(* CODESYS project GPS.4g.20210713.1.project

Project tree, tasks and I/O mapping:
  MIC7001 : Changsha-Cyber-MI-linux, Changsha Cyber-MI Co., Ltd., version 3.5.10.40
    application Application
      libraries: Standard, * (System); CAA Types Extern, * (CAA Technical Workgroup); CAA Callback Extern, * (CAA Technical Workgroup); SysMem, * (System); SysTypes Interfaces, * (System); SysTime, * (System); CAA DTUtil Extern, 3.5.12.0 (CAA Technical Workgroup); CAA Real Time Clock Extern, 3.5.10.0 (CAA Technical Workgroup); CAN API, 1.0.0.3 (3S - Smart Software Solutions GmbH); SysFile, 3.5.15.0 (System); AC_DataLog, 3.5.14.0 (3S - Smart Software Solutions GmbH); CAA Net Base Services, 3.5.15.0 (CAA Technical Workgroup); CAA Memory, 3.5.12.0 (CAA Technical Workgroup); CAA SerialCom, 3.5.15.0 (CAA Technical Workgroup); Util, 3.5.15.0 (System); CAA Can Low Level Imp Extern, 3.5.11.0 (CAA Technical Workgroup); CAA Can Low Level Extern, 3.5.15.0 (CAA Technical Workgroup); VisuDialogs, * (System); CmpBitmapPool, * (System); CAA File, 3.5.15.0 (CAA Technical Workgroup); IODrvEtherCAT, 3.5.15.50 (3S - Smart Software Solutions GmbH); SysShm Implementation, 3.5.16.0 (System); SysShm, 3.5.8.0 (System); MIC7001 base library, 1.11 (Cyber-MI.com)
      task VISU_TASK (cyclic, interval 100 ms, priority 31) calls prg_gps, VisuElems.Visu_Prg
      10_gvls/
        global variables gvl_remoter
        global variables GVL_prg_weight
        global variables GVL_IO
        global variables GVL_ES
        global variables GVL
        global variables GVL_can
        global variables GVL_par
      06_jt808/
        programs/
          program prg_gps [ST]
          program prg_jt808 [ST]: send_to_server, read_from_server, init
        Structs/
          data type stShmJT808Down
          data type stLocationExt
          data type stShmJT808Up
          data type stLocationBase
          data type stCanFrm
          data type nmeaTIME
          data type nmeaGPRMC
        functionblocks/
          function block Com_gps [ST]
        functions/
          function get_sub_string_1 [ST]
          function nmea_parse_time [ST]
          function nmea_parse_date [ST]
          function get_latlon_from_str [ST]
          function nmea_parse_GPRMC [ST]
    SoftMotion General Axis Pool
  libraries: CmpBitmapPool, * (System)
  5ce3da45-db07-42e7-a21c-a00fff4ed8f6|D:\工作文件\009中集集团\DOCS\等油耗图.jpg
  5ce3da45-db07-42e7-a21c-a00fff4ed8f6|C:\Users\RJST\Desktop\bmp1.png
  text list GlobalTextList
*)

// MIC7001/Application/06_jt808/Structs/stShmJT808Down
TYPE stShmJT808Down :  // JT808下行数据
STRUCT
	location_interval:DINT;  // 位置信息发送间隔， 单位： ms
	ctrl : DINT;   // 车辆控制命令
END_STRUCT
END_TYPE

// MIC7001/Application/06_jt808/Structs/stLocationExt
TYPE stLocationExt :
STRUCT
	km_all: DINT;  // km all
	fuel:INT;   // fuel meter
	speed: INT;  // speed can
	lac:DINT; 
	cid:DINT;
	fuel_trip:DINT; // 本行程油耗
	fuel_all:DINT; 
	fuel_r_h:DINT;  // 0.05L/h
	fuel_r_l:DINT;  //  1/512Km/L
END_STRUCT
END_TYPE

// MIC7001/Application/06_jt808/Structs/stShmJT808Up
TYPE stShmJT808Up :   // 发送到服务器的上行数据
STRUCT
    location:stLocationBase;
	loc_ext:stLocationExt;
	can_data:stCanFrm;
END_STRUCT
END_TYPE

// MIC7001/Application/06_jt808/Structs/stLocationBase
TYPE stLocationBase :
STRUCT
	warning : UDINT;
    status : UDINT;
    latitude : DINT;
    longitude : DINT;
    altitude : INT;
    speed : INT;
    bearing : INT;
    asc_time :ARRAY[0..5] OF BYTE;  // ascii YYMMDDhhmmss (GMT+8)
END_STRUCT
END_TYPE

// MIC7001/Application/06_jt808/Structs/stCanFrm
TYPE stCanFrm :
STRUCT
	sn:UDINT;  // 每次更新内容后加一，用于通知底层发送程序
	id:UDINT;  //  CAN id
	data:ARRAY[0..7] OF BYTE;  // 8个字节 数据
END_STRUCT
END_TYPE

// MIC7001/Application/06_jt808/Structs/nmeaTIME
TYPE nmeaTIME :
STRUCT
	year:DINT;
	month:DINT;
	day:DINT;
	hour:DINT;
	minute:DINT;
	second:DINT;
	hsecond:DINT;
END_STRUCT
END_TYPE

// MIC7001/Application/06_jt808/Structs/nmeaGPRMC
TYPE nmeaGPRMC :
STRUCT
	utc : nmeaTIME;
	status : STRING(1);
	lat : REAL;
	ns : STRING(1);
	lon : REAL;
	ew : STRING(1);
	speed : REAL;
	direction : REAL;
	declination : REAL;
	declin_ew : STRING(1);
	mode : STRING(1);
END_STRUCT
END_TYPE

// MIC7001/Application/10_gvls/gvl_remoter
{attribute 'qualified_only'}
VAR_GLOBAL
    // byte0
    link:DINT;   //连接状态
    acc: BOOL ;  // 加速
    dec:BOOL ;   // 减速
    mix:BOOL;    // 搅拌
    dump:BOOL;   // 卸料
    
    // byte1
    up:BOOL;     // 
    down:BOOL;
    left:BOOL;
    right:BOOL;
    auto_add_water:BOOL;
    e_stop:BOOL;  // 急停按钮
    
    // byte2
    
END_VAR

// MIC7001/Application/10_gvls/GVL_prg_weight
{attribute 'qualified_only'}
VAR_GLOBAL
	
weight_01,weight_02,weight_03:REAL:=0;

weight_load_01,weight_load_02,weight_load_03:REAL:=0;

net_weight:REAL:=0;


ad_load	 :REAL; 
SET_load1   :REAL;  	//设定重量 砝码1
SET_load2   :REAL;	//设定重量 砝码2
SET_load3 	:REAL;		//设定重量 砝码3
SET_load4   :REAL;  	//设定重量 砝码1
SET_load5   :REAL;	//设定重量 砝码2
SET_load6 	:REAL;		//设定重量 砝码3

load_up1    :REAL;	//标定的提升重量 1
load_up2   :REAL;		//标定的提升重量 2
load_up3 	:REAL;;		//标定的提升重量 3
load_up4    :REAL;	//标定的提升重量 1
load_up5   :REAL;		//标定的提升重量 2
load_up6 	:REAL;;		//标定的提升重量 3


AD_load_up1    :REAL;
AD_load_up2    :REAL;
AD_load_up3    :REAL;
AD_load_up4    :REAL;
AD_load_up5    :REAL;
AD_load_up6    :REAL;


END_VAR

// MIC7001/Application/10_gvls/GVL_IO
{attribute 'qualified_only'}
VAR_GLOBAL

AI_curr_a				:   DWORD ;   	// 电磁阀电流A
AI_curr_b				:   DWORD ;   	// 电磁阀电流B

Putter_position			:   DWORD ;     // C17推杆位置
A_three_load			:	DWORD;		// C29 三态开关信号

AI_F_Tank_speed_set		:   DWORD ;  	//	C31 /角位移 前面罐速设定
AI_BL_Tank_speed_set	:   DWORD ;   	//  C19 后左罐速设定
AI_BR_Tank_speed_set	:   DWORD ;   	//  C20后右罐速设定

Joystick				:	DINT;   // 操纵杆 角位移
set_speed_Tank			:	REAL;	//设定罐子速度
Joystick_min			:	DINT:=2020 ; 	//小值
Joystick_mid			:	DINT :=2405; 	//中值
Joystick_max			:	DINT :=2642; 	//最大值



set_speed_temp_tank		:	real;	// 设定罐速

VCC						:   DWORD ;		//控制电压
VCC_L					:   DWORD ;		//系统电流
A_REMOTe_youmen			:   DWORD ;		//远程油门
out5v			:   DWORD ;		//输出5V 
AI_Putter_position_feedbake	:   DWORD:=0 ;		// C17 阀推杆位置反馈


// out 
bforeward_Direction		:	BOOL;		//C03 搅动指示 
bRevers_Direction		:	BOOL;		// C01 出料状态指示灯 
 
out_tor_grade_k1		:BOOL;		 	//  C25  中载  多态输出K1
out_tor_grade_k2		:BOOL; 			//  C24	 轻载 多态输出K2

hb_pwm_L				:DWORD:=0;		//  C08电机正转 输出电流
hb_do_L					:BOOL:=FALSE;	//  C23电机正转 H桥低有效

hb_pwm_R				:DWORD:=0;		//  C09电机反转 输出电流
hb_do_R					:BOOL:=FALSE;	//  C35电机反转  H桥低有效
	
/////////////////////////
pwmForward 				: DWORD;  		// 
pwmRevers 				: DWORD;  	 	// 

Pump_foreward			:	DWORD ;     // 泵比例1 正转
Pump_Revers			:	DWORD;  // 泵比例2 反转
Throttle 		:	DWORD;   // 远程油门  0.3 ~ 1.9V
Throttle2 		:	DWORD;   // 远程油门 2 倍  0.6 ~ 3.8V






//Tank_dir			:	BOOL;  //计数 A
Tank_Speed_count		:	DWORD;  //计数 B
//bWater_washlimt	: 	BOOL; // 摆杆限位 

PI02_A,PI03_B:DWORD;		//接近开关计数
PI00,PI01,PI02,PI03	:DWORD;	//接近开关计数

DI02_A,DI03_B	: 	BOOL; 	//接近开关电平



lagan_foreward_Direction		:	BOOL;	//拉杆搅动
lagan_Revers_Direction		:	BOOL;	// 拉杆 卸料

//b_foreward_Direction	:	BOOL;	//搅驾驶室操作搅动
//b_Revers_Direction		:	BOOL;	//驾驶室操作 卸料




remote_di :BOOL := FALSE; //绑定变量 驾驶室开关， 为True则通过遥控方式控制罐体， 不使用拉杆
b_mode_remote : BOOL  := FALSE;  // 驾驶室开关， 为True则通过遥控方式控制罐体， 不使用拉杆


SET_Putter_position:DINT;	//推杆位置 换算
Putter_avg:	DINT;		//推杆位置 
Putter_mid_dema:	DINT;//推杆中位标定
Putter_position_ERR,Joystick_ERR,J1939_ERR	:BOOL; //角位移，电机位置反馈  故障指示
flag_stir_enable:BOOL	;//允许搅动状态位
flag_Constant_speed:BOOL	;// 不允许 卸料 标志位 

//处理之后的数值

temp_Hydraulic_oil:REAL;	//油温值
Dprss_pumpA		:REAL; 		//正转马达压力值
Dprss_pumpB		:REAL; 		//反转马达压力值
Dprss_Water		:REAL;		//清洗水压
Dwater_level	:REAL;		//水位

iPump_foreward		:	REAL;   // 泵比例正向 
iPump_Revers 		:	REAL;  	// 泵比例反向
itank_dir            :DINT;
iPump_PID            :REAL;
END_VAR

// MIC7001/Application/10_gvls/GVL_ES
{attribute 'qualified_only'}
VAR_GLOBAL
	// send to cloud my mqtt	
	working_mode:UINT;  // 工作模式 0:熄火停车， 1：空车等待， 2：正在装料， 3：满车行驶，4：满车等待，5：正在卸料， 6：空车行驶
	rpm_engine:DINT; // 发动机转速  转/分
	rpm_set :DINT ;  // 设定发动机转速 转/分
	power_engine:REAL; // 发动机功率 千瓦
	torque_engine:REAL;// 发动机扭矩 牛米
	fuelrate_engine:REAL;// 发动机瞬时油耗 升/小时
	effect_engine:REAL;// 发动机瞬时效率 %
	fuelall_engine:REAL;// 发动机累计油耗 升
	loadrate_engine:REAL;// 发动机负载率 %
	hours_engine:REAL;// 发动机工作时间  小时
	press_pump:REAL; // A B 口压力差
	press_pump_a:REAL;// 油泵主压 A 兆帕
	press_pump_b:REAL;// 油泵主压 B 兆帕
	dir_pump:DINT;// 油泵方向 1：正转， 0： 停止，  -1：反转
	curr_a_pump:REAL;//  油泵电流A  毫安
	curr_b_pump:REAL;//  油泵电流B  毫安
	power_pump:REAL;// 油泵输出功率 千瓦
	swept_pump:REAL;// 油泵排量 毫升/转
	flow_pump:REAL;// 油泵流量 升/分
	effect_pump:REAL;// 油泵效率 %
	torque_pump:REAL;// 油泵扭矩 牛米
	dir_tank:DINT;// 搅拌桶方向 1：正转， 0： 停止，  -1：反转
	rpm_tank:REAL;// 搅拌桶转速 转/分
	weight_tank:REAL;// 搅拌桶重量 吨
	power_tank:REAL;// 搅拌桶功率 千瓦
	effect_tank:REAL;// 搅拌桶效率 %
	torque_tank:REAL;// 搅拌桶扭矩 牛米
	volume:REAL;// 当前方量 立方米
	volume_all:REAL;// 累计方量 立方米
	mileage_all:REAL;// 累计里程 千米
	grade_gear:DINT;// 变速箱档位
	rate_gear:REAL;// 变速箱变比
	rpm_gear:REAL;// 变速箱输出转速 转/分
	torque_gear:REAL;// 变速箱输入扭矩 牛米
	power_gear:REAL;// 变速箱输出功率 千瓦
	effect_gear:REAL;// 变速箱效率 %
	weight_all:REAL;// 整车重量 吨
	speed:REAL;   // 行车速度 Km/h
	power_running:REAL;  // 行车功率 Kw
	acc_running:REAL; // 行车加速度 Km/h/s
	fuel_trip_engine:REAL;  // 行程总油耗
	torque_grade:DINT;  // 节能模式： 0：轻载， 1： 中载，  2：重载
	acc_pad : REAL;  // 油门踏板 百分比
	fuel_wait:REAL :=0;  // 本行程等待油耗 L
    time_wait:REAL := 0;  // 本行程等待时间 s
    fast_acc_cntr :DINT := 0; // 急加速次数
    fast_dec_cntr :DINT := 0; // 急刹车次数
    low_grade_cntr:DINT := 0; // 低档高速次数
	fuel_100km:REAL;  // 百公里油耗
    fuel_level:REAL;  // 油耗水平 0~100
	Engine_Hour:REAL;
	
	trip_all_1939:REAL;    // 里程累计
	trip_curr_1939:REAL;  // 里程小计

	trip_all_1939_2:REAL;    // 里程累计, 高分辨率
	trip_curr_1939_2:REAL;  // 里程小计, 高分辨率
	
	temp_coolant_1939:DINT;
	Eng_Fuel_Temp:DINT;
	Eng_Oil_Temp:DINT;
	Turbo_Oil_Temp:DINT;
	Eng_InterCooler_Temp:DINT;
	Eng_InterCooler_Thermostat_Opening:DINT;
	oil_press_1939:REAL;
	coolant_level_1939:REAL;
	acc_set:BYTE;
    
    rpm_disp:ARRAY[0..9999] OF DINT;
    tor_disp:ARRAY[0..9999] OF DINT;
    ptr_disp:DINT  := 0;
    x:DINT;
    y:DINT;
    z:DINT;
	grade_joystick:REAL := 0;  // 1~10
	
	shift:DINT;  // 离合
	brake:DINT;  // 刹车
END_VAR

VAR_GLOBAL CONSTANT
	retain_max : DINT := MIC7001_BASE.Constants.RETAIN_NUM_MAX;
	// 柴油机扭矩曲线
	rpm_in:ARRAY[0..255] OF REAL := [700, 800,  900,  1000, 1100, 1200, 1300, 1400, 1500, 1600, 1700, 1800, 1900, 2000, 2100];
 	tor_h:ARRAY[0..255] OF REAL :=  [922, 1100, 1350, 1488, 1600, 1600, 1600, 1600, 1570, 1495, 1410, 1320, 1221, 970,  555];
	tor_m:ARRAY[0..255] OF REAL :=  [922, 1100, 1350, 1488, 1600, 1550, 1480, 1350, 1200, 1000,  750, 0,     0,   0,    0];
 	tor_l:ARRAY[0..255] OF REAL :=  [922, 1100, 1200, 1020, 800,  620,  460,  320,  200,  100,   0,   0,     0,   0,    0];	
END_VAR

// MIC7001/Application/10_gvls/GVL
VAR_GLOBAL CONSTANT
	retain_max : DINT := MIC7001_BASE.Constants.RETAIN_NUM_MAX;
END_VAR

VAR_GLOBAL
	
	flag_mode:bool;
	bTank_wash_Fnish:BOOL;
	
	xEnaSE:BOOL := TRUE;  // 启用节能模式
	xEnaLowRPM:BOOL := TRUE;  // 启用起步降速功能
	xEnaTor :BOOL := TRUE;  // 启用扭矩调节功能
	
	//熟数据
	g_ai_press_pump : REAL;  // 油泵主压， 单位： MPa	
	
	falg_tank_control,flag_chute_control,flag_Clean_control:BOOL;
	
	//
	g_uiYear:UINT := 1970;
	g_uiMonth:UINT := 1;
	g_uiDate:UINT := 1;
	g_uiHour:UINT := 0;
	g_uiMinute:UINT := 0;
	g_uiSecond:UINT := 0;
	
	//小时计相关
	g_running_mins:DINT := 0; //控制器运行的分钟数  retain
	g_engine_mins:DINT := 0; //发动机运行的分钟数   retain
	
	g_engine_mins_1_start:DINT := 0; //阶段小时计1开始时间  retain
	g_engine_mins_2_start:DINT := 0; //阶段小时计2开始时间  retain

	g_engine_mins_1:DINT := 0;  //发动机运行分钟数  阶段1 
	g_engine_mins_2:DINT := 0;  //发动机运行分钟数  阶段2
	
	// PORT CAN1 GLOBAL HANDLE
	g_hCan1939: CAA.HANDLE ;
	g_hRecv_FEEE: CAA.HANDLE := 0;
	g_hRecv_FEEF: CAA.HANDLE := 0;
	g_hRecv_F003: CAA.HANDLE := 0;
	g_hRecv_F004: CAA.HANDLE := 0;
	g_hRecv_18F: CAA.HANDLE := 0;
	
	//发动机相关实时数据
	g_P_KW_max:DINT := 30;  //当前发动机储备功率
	g_rpm_set: DINT := 1000;  //当前设定转速
	g_rpm_real: DINT := 0; //当前实时转速
	g_fuel_rate_1939:REAL := 0; //从发动机读到的瞬时油耗，单位：ml/s
	g_temp_coolant_1939:REAL := 0; //从发动机读到的水温， 单位：摄氏度
	g_flag_coolant_high:bool := false;  //水温报警标志
	g_oil_press_1939:REAL := 0; //从发动机读到的机油压力， 单位： kPa
	g_coolant_level_1939:REAL := 0; //从发动机读到的冷却液液位， 单位： 百分比
	g_load_percent_1939:REAL := 0; //从发动机读到的发动机负载率， 单位： 百分比
	g_demand_torque_1939:DINT := 0; //从发动机读到的需求扭矩， 单位： 百分比
	g_real_torque_1939:DINT := 0; //从发动机读到的实际扭矩， 单位：百分比
	g_acc_1939: BYTE := 0;  //从发动机读到的油门踏板百分比
	g_perfect_rpm: DINT := 0;  //从发动机读到的当前理想转速，单位 ：rpm
	g_tor_idle_1939: BYTE := 0;  //从发动机读到的当前摩擦转矩，单位：百分比
	g_real_torque_nm_1939: DINT := 0;
	g_working_old:BOOL := FALSE;
//动态调整参数	


	g_acc_set :BYTE := 40;   //需要设置的油门踏板百分比
	g_tor_set :BYTE := 1;   //需要设置的扭矩曲线号
	g_droop_set :BYTE := 16#F0;   //设置调速率

	rpm_lost_point:DINT := 50;
	
	g_x_duty_max :REAL := 70;	
	g_x_duty_min :REAL := 60;
	g_x_rpm_up_step: INT := 5;
	g_x_rpm_down_step: INT := 1;
	
	g_x_tor_max:REAL := 90;
	g_x_tor_min:REAL := 70;
	g_x_pump_up_step: INT := 1;
	g_x_pump_down_step: INT := 2;
	
	g_enable_rpm_adj:BOOL := TRUE;
	

	//retain paras 
	g_retain_01:ARRAY[0..retain_max] OF DINT;
	g_retain_02:ARRAY[0..retain_max] OF DINT;
	g_mins:ARRAY[0..MIC7001_BASE.Constants.RETAIN_NUM_MAX] OF DINT;
//动态调整参数	
	
	//统计数据
	g_fuel_depleted : DINT := 0;  //出厂累计油耗，单位：毫升
	g_fuel_depleted_1: DINT := 0; //阶段一累计油耗，单位：毫升
	g_fuel_depleted_2: DINT := 0; //阶段二累计油耗，单位：毫升
	
	g_Eng_Coolaant_Temp:INT;(*spn 110*)
	g_Eng_Fuel_Temp:INT;(*spn 174*)
	g_Eng_Oil_Temp:INT;(*spn 175*)
	g_Turbo_Oil_Temp:INT;(*spn 176*)
	g_Eng_InterCooler_Temp:INT;(*spn 52*)
	g_Eng_InterCooler_Thermostat_Opening:BYTE;(*spn 1134*)
	
						
	g_res_prop:REAL := 20; //电磁比例阀电阻，动态调整

	g_ai_pilot:REAL;
	g_ai_pilot_trace: REAL;
	g_ai_curr_prop:UINT;
	g_ai_curr_prop_trace:REAL;
	g_ai_oil_water:BOOL;
	g_ai_vcc:DWORD;
	g_ai_fuel_level:REAL;

	g_di_start:BOOL := FALSE; //上电信号
	g_di_move:BOOL := FALSE; //工作装置压力开关
	g_di_work:BOOL := FALSE; //行走压力开关
	g_di_pilot:BOOL := FALSE;  //先导手柄开关输入
	
	g_do_start:BOOL := TRUE;  //启动继电器		
	g_do_ecu:BOOL := TRUE;    //为true为发动机ECU供电
	g_do_pilot:BOOL := FALSE;
	
	g_pwm_prop:DINT := 0; 
	
	g_rpm_trace:REAL := 0;  //示波器变量，转换到0~10之间
	//间接计算数据
	g_psp: REAL := 0;   //电磁比例阀二次压力  MPa
	g_backup_power:REAL := 0;   //发动机储备功率  KW
	g_backup_power_trace:REAL; //示波器变量，转换到0~10之间
	g_duty_power:REAL := 0; //发动机功率利用率
	g_backup_torque:REAL := 0;  //发动机储备扭矩  N*M
	g_backup_torque_trace:REAL;//示波器变量，转换到0~10之间
	g_duty_torque:REAL := 0;  //发动机扭矩利用率
	g_flow1 :REAL := 0;   //前泵流量 L/min
	g_flow1_trace:REAL;//示波器变量，转换到0~10之间
	g_flow2 :REAL := 0;   //后泵流量 L/min
	g_flow2_trace:REAL;//示波器变量，转换到0~10之间
	g_power_pump1 :REAL := 0;   //前泵功率  KW
	g_power_pump1_trace:REAL;//示波器变量，转换到0~10之间
	g_power_pump2 :REAL := 0;   //后泵功率  KW
	g_power_pump2_trace:REAL;//示波器变量，转换到0~10之间
	g_torque_pump1 :REAL := 0;  //前泵输出扭矩  N*M
	g_torque_pump2 :REAL := 0;  //后泵输出扭矩  N*M
	
// I/O port mapping var
	AI_pump1:DWORD; //前泵压力
	AI_pump2:DWORD; //后泵压力
	AI_pilot:DWORD; //先导压力
	AI_curr_prop:DWORD; //电磁比例阀电流
	AI_oil_water:DWORD; //油水分离器
	AI_vcc:DWORD; //电源电压 mV
	AI_grade:DWORD; //油门旋钮
	AI_temp_oil:DWORD; //液压油温
	AI_fuel_level:DWORD; //液位传感器
	AI_idle_button:dword; //机械怠速按钮
	
	DI_start: BOOL; //启动信号
	DI_pilot:BOOL; //先导手柄闭合
	DI_move:BOOL; //行走压力开关
	DI_work:BOOL; //作业压力开关
	DI_air_filter:BOOL;  //空滤堵塞
	DI_idle_button:BOOL;  //机械怠速按钮
	DI_high_power:BOOL; //增力信号输入
	
	DO_start: BOOL := FALSE; //驱动启动电机
	DO_stop: BOOL := TRUE;  //驱动熄火继电器
	DO_pilot :BOOL := TRUE;  //驱动先导阀
	DO_high_power:BOOL := FALSE; //增力输出
	DO_high_speed:BOOL := FALSE; //高速输出
	DO_dump_load:BOOL := FALSE; //卸载输出
						
	PWM_prop:DWORD; //油泵电磁比例阀	
	
	RPM_engine:UINT; //柴油机转速  J1939

	DO_led_run:BOOL;
	DO_led_err:BOOL;
	DO_led_usr:BOOL;
	
// 档位校准	
	adj_gear: BOOL := FALSE;  //校准档位旋钮
	gear_grade: UINT := 1;   //档位旋钮对应的档位
	running_grade:DINT := 1;  //当前实际运行的档位
	
	g_grade: DINT;	  //发动机档位
	//各档位对应的转速

	g_running_grade_x:DINT := 1;
	g_power_avg_num: DINT := 10;  // 200 ms
	g_method_mode_A :DINT := 0;   // 0: based power_avg;   1: based load1939
	g_overpress_time:DINT := 100;   //1 second
	
//显示屏发送来的命令
//	cmd_auto_idle : BOOL := TRUE;
//	cmd_high_speed: BOOL := FALSE;	
//	cmd_more_power: BOOL := FALSE;
//	cmd_clear_hours : BOOL := FALSE;
//	cmd_clear_hours_1 :BOOL := FALSE;
//	cmd_clear_hours_2 :BOOL := FALSE;
	
	g_time_good: BOOL := FALSE;  //控制器本地时钟校准完成
	g_working: BOOL := false;
	g_err_fuel_level: BOOL;
	g_fuel_level: DINT;
	adj_1: BOOL;
	adj_10: BOOL;
	
	rpm_lost_rate: REAL;
	g_err_temp_oil: BOOL;
	g_temp_oil: DINT := 0;


	
	g_duty_power_avg: REAL := 0;
	g_duty_torque_avg: REAL;

	g_x_power_avg: REAL := 0;
	g_x_dest_grade: DINT := 1;
	g_torque_engine: REAL := 0;
	g_power_engine: REAL := 0;
	mode_a_up: DINT := 90;   // %
	mode_a_down:DINT := 80;  // %
	g_press12_avg: REAL := 0;
	g_press12_avg_all: REAL := 0;
	g_fuel_all_1939: DINT := 0;
	g_fuel_all: DINT := 0;
	
	g_lock_flag:BOOL := FALSE;
	g_lock_level:DINT := 0;
	gps_lock_h: BOOL := FALSE;
	gps_lock_s: BOOL := FALSE;
	gps_lock_l: BOOL := FALSE;
	
	need_send_mid :ARRAY[16#507..16#520] OF BOOL;
	need_ack_mid :ARRAY[16#307..16#320] OF BOOL;
	got_ack_mid :ARRAY[16#307..16#320] OF BOOL;
	
END_VAR




(*end of var_global for mqtt *****************************************************)


VAR_GLOBAL CONSTANT
	inmode_file:STRING:='/userapp/PlcLogic/in_mode.txt';
	mins_file :STRING := '/userapp/r_mins.txt';
END_VAR

// MIC7001/Application/10_gvls/GVL_can
{attribute 'qualified_only'}
VAR_GLOBAL
	
//can_send

	g_acc_set:BYTE;
	g_tor_set:BYTE; //扭矩曲线选择，0对应最高，2对应最低
	g_droop_set:BYTE;

	CansendData_18FF01FF : ARRAY[0..7] OF BYTE;     //系统传感器ID（搅拌车）0x18FF01FF  T 100ms   控制器发送 	
	
	CansendData_18FF02FF : ARRAY[0..7] OF BYTE;     //系统传感器ID（搅拌车）0x18FF01FF  T 100ms   控制器发送 	
	CansendData_18FF03FF : ARRAY[0..7] OF BYTE;     //系统传感器ID（搅拌车）0x18FF01FF  T 100ms   控制器发送 	
	
	CansendData_18FF66FF : ARRAY[0..7] OF BYTE;     //智能自动化控制器ID1（搅拌车）	0x18FF66FF	65280	6	Periodic	500 SEND 
	CansendData_18FF68FF : ARRAY[0..7] OF BYTE;  //智能自动化控制器报警ID1（搅拌车）	0x18FF68FF	65280	6	Periodic	500ms

	
	
	LoadingWashST,UnloadingWashReqST :BOOL;
	AutoClearWaterReqST:BOOL;
	AutoAddWaterReqST:BOOL;
	TankWashReqST:BOOL;
//can_receive
	
	CanReadData_18FF46FF : ARRAY[0..7] OF BYTE; 	//塌落度 ID 0x18FF46FF   T 500ms   网关发送 	
	CanReadData_18FF61FF : ARRAY[0..7] OF BYTE; 	//胎压传感器数据帧ID 0x18FF61FF  T 250ms   网关发送    暂不接收和转发
	CanReadData_18FF62FF : ARRAY[0..7] OF BYTE; 	//自动充气ID 0x18FF62FF   T 250ms   网关发送    暂不接收和转发	
	CanReadData_18FF64FF : ARRAY[0..7] OF BYTE;		//集中润滑ID	0x18FF64FF	65280	6	Periodic	500  网关发送    暂不接收和转发
	CanReadData_18FF6AFF : ARRAY[0..7] OF BYTE;		//GW_AdasInputs2	ADAS系统输入信息  ID2	0x18FF6AFF	65280	6	Periodic	100 网关  无用
	
	CanReadData_18FF01FE : ARRAY[0..7] OF BYTE;		//HU_ControlInformation1	大屏 ID1	0x18FF01FE	65280	6	Periodic	100	8  
	CanReadData_18FF02FE : ARRAY[0..7] OF BYTE;		//HU_ControlInformation2	大屏ID2		0x18FF02FE	65280	6	Periodic	100ms	8  FROM 显示屏据
	CanReadData_18FF03FE : ARRAY[0..7] OF BYTE;		//HU_ControlInformation2	大屏ID3		0x18FF03FE	65280	6	Periodic	100ms 	8  FROM 显示屏据

demo_cntr:UINT := 0;

// 控制器发送到操作面板数据 0x18ff01ff
CS_act_TankRPM 					:BYTE;		//	罐体转速			1.1 	8	0-20R/MIN
CS_set_TankRPM 					:BYTE;		//	设置转速			2.1 	8	0-20R/MIN
CS_TankRotateDirection			:BYTE;		//	放向			   3.1 	    2	0-20R/MIN
CS_Eenginespeed                  :dint;		// 发动机转速  		   4.1     16 rpm
CS_pump_press_A                  :BYTE;		// 泵压力  			   6.1     8   bar
CS_LiquidTemperature		     	:BYTE;		//	液压温度		   7.1		8	0~120°
// 控制器发送到操作面板数据 0x18ff02ff  
CS_STOPtank_warning		    	:BOOL;		//	罐体停止			1.1 	1	
CS_pump_pressA_warning 			:BOOL;		//	泵A压力故障			1.2 	1	
CS_pump_pressB_warning 			:BOOL;		//	泵B压力故障			1.3 	1	
CS_LiquidTemperature_warning     :BOOL;      //温度报警				1.4     1
CS_water_press_warning 			:BOOL;       //水压力报警      		1.5
CS_Water_level_warning			:BOOL;       //水位报警            	1.6
CS_Water_full_warning			:BOOL;       //水位报警            	1.7
CS_Water_miss_warning			:BOOL;       //水位报警            	1.8
CS_hightemp_warning 			:BOOL;       //高温报警				2.1
CS_Chute_warning 				:BOOL;       //出料槽故障			2.2
CS_addwater_warning 			:BOOL;       //加水清水故障				2.3

CS_Watet_press                  :BYTE;       // 水压					3.1    8
CS_Water_level                  :BYTE;		// 水位					3.2	   8
// 控制器发送到操作面板数据 0x18ff03ff  
CS_Work_Status      			:BOOL;      //工作指示灯           1.1    1
CS_Work_stop_Status      		:BOOL;      //状态指示灯           1.2    1
CS_Work_warning    				:BOOL;      //异常指示灯           1.3    1
CS_addspeed_Status       		:BOOL;      //加速指示灯           1.4    1
CS_decspeed_Status      		:BOOL;      //减速指示灯           1.5    1

CS_model_startStatus   		  	:BOOL;      //z装卸料启停          1.6    1
CS_model_pavingStatus   	   	:BOOL;      //铺路模式状态         1.7    1
CS_model_LoadStatus_H  		   	:BOOL;      //z装卸恒速 状态       1.8    1
CS_model_unloadStatus_H   	   	:BOOL;      //z卸料恒速状态        2.1    1
CS_model_LoadStatus   		   	:BOOL;      //z装卸 状态           2.2    1
CS_model_unloadStatus   	   	:BOOL;      //z卸料状态            2.3    1
CS_model_Chute_startStatus 	   	:BOOL;      //出料槽启动状态       2.4    1
CS_model_ChuteresetStatus  	   	:BOOL;      //出料槽复位状态       2.5    1
CS_model_Chute_upStatus   	   	:BOOL;      //出料槽上状态         2.6    1
CS_model_Chute_dowStatus  	   	:BOOL;      //出料槽下状态         2.7    1
CS_model_Chute_leftStatus      	:BOOL;      //出料槽左状态         2.8    1
CS_model_Chute_rigStatus  	   	:BOOL;      //出料槽右状态         3.1    1

CS_AI_curr_a			        :   DINT ;   // 电磁阀电流A
CS_AI_curr_b			        :   DINT ;   // 电磁阀电流B
CS_pump_press_b                  :BYTE;		// 泵压力  			   6.1     8   bar
// 操作面板发送到控制器的命令 0x18ff01fe  
CR_ADD_tankspeed                :BOOL; //罐体加速                  2.1    1
CR_dec_tankspeed                :BOOL; //罐体减速                  2.2    1
CR_model_start   		    	:BOOL;      //z装卸料启停          2.3   1
CR_model_paving			   	   	:BOOL;      //铺路模式       	   2.4    1
CR_model_Load_H  	     	   	:BOOL;      //z装卸恒速       	   2.5    1
CR_model_unload_H   	    	:BOOL;      //z卸料恒速      	   2.6    1
CR_model_Load        		   	:BOOL;      //z装卸                2.7    1
CR_model_unload         	   	:BOOL;      //z卸料            	   2.8    1
CR_model_Chute_start	 	   	:BOOL;      //出料槽启动           3.1    1
CR_model_Chutereset		  	   	:BOOL;      //出料槽复位           3.2    1
CR_model_Chute_up		   	   	:BOOL;      //出料槽上             3.3    1
CR_model_Chute_doW		  	   	:BOOL;      //出料槽下             3.4    1
CR_model_Chute_left		      	:BOOL;      //出料槽左             3.5    1
CR_model_Chute_rig       	   	:BOOL;      //出料槽右             3.6    1
CR_model_ADDwater_start       	:BOOL;      //出料槽右             4.1    1
CR_model_ADDwater		      	:BOOL;      //出料槽右             4.2    1
CR_model_diswater		      	:BOOL;      //出料槽右             4.4    1
CR_model_lamp_switch	      	:BOOL;      //出料槽右             5.2    1





























//系统传感器ID（搅拌车）0x18FF01FF  T 100ms   控制器 发送 
LiquidTemperature			:BYTE;		//	液压温度			1	0	8	0~120°
TankRotateDirection			:BYTE;		//	罐体转动方向		2	8	2  0-停止 1-正转  2-反转
LiquidTemperatureWarning	:BYTE;		//	液压温度报警状态	2	10	1	"0-正常 1-报警"
//Reserved 									 		保留		2	11	5	
TankRPM 					:BYTE;		//	罐体转速			3	16	8	0-20R/MIN

//塌落度 ID 0x18FF46FF   T 500ms   网关发送 
SLUMP						:DINT;		//	塌落度				1	0	16	mm
//TankRPM						:BYTE;		//	罐体转速			3	16	8	TankRPM*0.1(R/min)
W_C							:BYTE;		//	水灰比				4	24	8	(W/C)/250
Formula						:BYTE;		//	配方				5	32	7	平台在前面加C(例C100)
SLUMPStatus					:BOOL;		//	塌落度故障状态		5	39	1	"0-正常   1-异常"
SLUMP_T						:DINT;		//	温度				6	40	8	(SLUMP-T)-40(摄氏度)
ResidualVolume				:DINT;		//	残余容积			7	48	16	L

//胎压传感器数据帧ID 0x18FF61FF  T 250ms   网关发送    暂不接收和转发

//自动充气ID 0x18FF62FF   T 250ms   网关发送    暂不接收和转发

//集中润滑ID	0x18FF64FF	65280	6	Periodic	500  网关发送    暂不接收和转发


//智能自动化控制器ID1（搅拌车）	0x18FF66FF	65280	6	Periodic	500 SEND 

WaterLevel				:BYTE;		//	水箱液位			1	0	8	0-195mm
AutoWaterStatus			:BYTE;		//自动加水状态			3	16	2	"0-初始  1-加水中  2-结束  3-异常"  
InHopperWashStatus		:BYTE;		//进料斗清洗状态		3	18	2	"0-初始 1-清洗中 2-结束 3-异常"
TankWashStatus			:BYTE;		//罐体清洗状态			3	20	2	"0-初始  1-清洗中 2-结束 3-异常"
OutHopperWashStatus		:BYTE;		//出料斗清洗状态		3	22	2	"0-初始 1-清洗中2-结束 3-异常"
TankWaterStatus			:BYTE;		//水箱清水状态			4	24	2	"0-初始 1-清水中 2-结束 3-异常"
TankSpeedMode			:BYTE;		//	罐速控制模式		4	26	3	"0-装料 1-运输 2-卸料3-铺路 4-零速"
WaterLevelWarning		:BOOL;		//	水箱液位低报警状态		4	29	1	非0报警
OutHopperPositionAdjustFB	:BYTE;	//	出料口位置调节反馈		4	30	2	"0-停止 1-运行中 2-左调节超时 3-右调节超时"
ControlModeFB				:BYTE;	//	智能控制方式反馈		5	32	2	"0x0:无效 0x1:车载屏控制   0x2:面板控制  0x3:APP控制"
GoHomeStatus				:BOOL;	//	搅拌车一键复位状态反馈	5	37	1	"0: 停止 1:复位中"
AutoDischargeStatus			:BYTE;	//智能自动卸料状态			6	40	2	"0-初始 1-卸料中2-结束3-异常"
EmergencyOffWarning			:BOOL;	//紧急熄火报警状态			6	42	1	"0-正常 1-异常"
OverPressureWarning1		:BOOL;	//超压报警状态				6	43	1	"0-正常1-异常"
OverPressureWarning2		:BOOL;	//近压报警状态				6	44	1	"0-正常1-异常"
//ControlModeFB				:BYTE; 	//智能控制方式反馈		7	50	2	"0x0:无效 0x1:车载屏控制 0x2:面板控制 0x3:APP控制"
Reserved					:BYTE; 	//保留					7	54	2	
//ControlModeFB				:BYTE; 	//	智能控制方式反馈		4	24	2	"0x0:无效 0x1:车载屏控制 0x2:面板控制 0x3:APP控制"

//智能自动化控制器报警ID1（搅拌车）	0x18FF68FF	65280	6	Periodic	500ms

Warning1		:BOOL;	//	开启水箱气控阀（1，0）后气压达到标准大气压时间超时		1	0	1	"0-Inactive 1-Active"
Warning2		:BOOL;	//	开始加水到水满的时间超时								1	1	1	"0-Inactive 1-Active"
Warning3		:BOOL;	//	开启水箱气控阀（0，1）后气压达到0.4标准大气压时间超时	1	2	1	"0-Inactive 1-Active"
Warning4		:BOOL;	//	摆杆归位超时											1	3	1	"0-Inactive 1-Active"
Warning5		:BOOL;	//	RPM不符合需求，无法驱动罐体转动							1	4	1	"0-Inactive 1-Active"
Warning6		:BOOL;	//	清水动作时长时间处于水满状态							1	5	1	"0-Inactive 1-Active"
Warning7		:BOOL;	//	自动加水结束											1	6	1	"0-Inactive  1-Active"
Warning8		:BOOL;	//	自动加水紧急停止										1	7	1	"0-Inactive 1-Active"
Warning9		:BOOL;	//	进料斗清洗结束											2	8	1	"0-Inactive 1-Active"
Warning10		:BOOL;	//		进料斗清洗紧急停止									2	9	1	"0-Inactive 1-Active"
Warning11		:BOOL;	//		罐体清洗完毕，开始出料口清洗						2	10	1	"0-Inactive1-Active"
Warning12		:BOOL;	//		出料口清洗完毕										2	11	1	"0-Inactive1-Active"
Warning13		:BOOL;	//		罐体清洗紧急停止									2	12	1	"0-Inactive 1-Active"
Warning14		:BOOL;	//		出料口清洗紧急停止									2	13	1	"0-Inactive 1-Active"
Warning15		:BOOL;	//		自动清水完毕										2	14	1	"0-Inactive 1-Active"
Warning16		:BOOL;	//		自动清水紧急停止									2	15	1	"0-Inactive 1-Active"
Warning17		:BOOL;	//		伺服电机驱动到最大位置超时							3	16	1	"0-Inactive 1-Active"
Warning18		:BOOL;	//		装料时罐体正转速度达到W1超时						3	17	1	"0-Inactive 1-Active"
Warning19		:BOOL;	//		装料超时未人工停止									3	18	1	"0-Inactive 1-Active"
Warning20		:BOOL;	//		装料完成后降速至W2超时								3	19	1	"0-Inactive 1-Active"
Warning21		:BOOL;	//		装料完成，自动切换为运输状态						3	20	1	"0-Inactive 1-Active"
Warning22		:BOOL;	//		卸料时罐体反转速度达到W3超时						3	21	1	"0-Inactive 1-Active"
Warning23		:BOOL;	//		卸料超时未人工停止									3	22	1	"0-Inactive 1-Active"
Warning24		:BOOL;	//		卸料完毕罐体降速至0超时								3	23	1	"0-Inactive 1-Active"
Warning25		:BOOL;	//		卸料完成，罐体处于0转速								4	24	1	"0-Inactive 1-Active"
//Reserved	预留		4	25	7	
//Reserved	预留		5	32	8	
//Reserved	预留		6	41	8	
//Reserved	预留		7	48	8	
//Reserved	预留		8	56	8	
RightTurnLightStatus		:BOOL;	//右转向灯		1	0	1	"0-Inactive  1-Active"
LeftTurnLightStatus			:BOOL;	//左转向灯		1	1	1	"0-Inactive  1-Active"
GearShiftPosition			:BOOL;	// 档位			1	2	4	"0x0:Parking  0x1:Reverse 0x2:Neutral 0x3:D 0x4:D3 0x5:D2 0x6:L 0x7:M/S
																	//0x8:Reserved   0xD:Reserved   0xE:Unreliable 0xF:Invalid"
BrakePedalStatus			:BOOL;	// 	制动踏板状态		1	6	1	"0x0:invalid 0x1:valid" 
//Reserved	预留											1	7	1	预留
SteeringAngle				:DWORD;	//  方向盘转向角度		2	8	16	
VehicleSpeed				:DWORD; //	车速				4	24	16	
YawingRate					:DWORD; //	横摆速率			6	40	16	
ENG_SPEED					:DWORD; //发送机实时转速
//Reserved			 					预留				8	56	8	预留


//GW_AdasInputs2	ADAS系统输入信息  ID2	0x18FF6AFF	65280	6	Periodic	100 网关  无用

BSDSwitch					:BOOL;	// 		BSD开关		1	0	1	"0-Inactive 1-Active"
LDWSwitch					:BOOL;	// 		LDW开关		1	1	1	"0-Inactive 1-Active"
RCWSwitch					:BOOL;	// 		RCW开关		1	2	1	"0-Inactive 2-Active"
AVMSwitchStatus				:BOOL;	// 		AVM按键状态	1	3	2	"0x0:Inactive/Initial value 0x1:Press down 0x2:Lift up"
//Reserved					:BOOL;	// 预留				1	5	3	
XAxisPixel					:BYTE;	// X轴分辨率/触摸屏width		2	8	12	
YAxisPixel					:BYTE;	// Y轴分辨率/触摸屏hight		3	20	12	
XAxisPosition				:BYTE;	// 触屏X轴/x坐标				5	32	12	
YAxisPosition				:BYTE;	// 触屏Y轴/y坐标				6	44	12	
PanelStatus					:BOOL;	// 触摸屏状态					8	56	2	"0x0:Inactive/Initial value  0x1:Press down 0x2:Moving  0x3:Lift up"
//Reserved								预留						8	58	6	

//HU_ControlInformation1	大屏 ID1	0x18FF01FE	65280	6	Periodic	100	8  

LoadingWashReq				:BYTE;	//	装料清洗请求		1	0	2	"0x0:无效  0x1:停止 0x2:开始"
UnloadingWashReq			:BYTE;	//	卸料清洗请求		1	2	2	"0x0:无效  0x1:停止 0x2:开始"
TankWashReq					:BYTE;	//罐体清洗请求			1	4	2	"0x0:无效 0x1:停止 0x2:开始"
AutoAddWaterReq				:BYTE;	//自动加水请求			1	6	2	"0x0:无效  0x1:停止 0x2:开始"
AutoClearWaterReq			:BYTE;	//自动清水请求		 	2	8	2	"0x0:无效 0x1:停止0x2:开始"
TankSpeedInLoadingMode		:BYTE;	//罐速控制装料模式		2	10	5	"0x0:无效 0x3:3R/min 0x4:4R/min———— 0x13:19R/min"
Tank0SpeedGoBack			:BOOL;	//罐速控制零速返程		2	15	1	"0x0:无效  0x1:打开"
TankSpeedInUnloadingMode	:BYTE;	//罐速控制卸料模式		3	16	5	"0x0:无效  0x3:3R/min  0x4:4R/min 0x5:5R/min————  0x13:19R/min 0x14:20R/min"
TankSpeedInTransMode		:BYTE;	//罐速控制运输模式		4	24	5	"0x0:无效  0x3:3R/min 0x4:4R/min  0x12:18R/min ————  0x13~0x1F 预留"
OutHopperPositionAdjust		:BYTE;	//出料口位置调节信号	4	29	3	"0x0:无效  0x1:上调节  0x2:下调节  0x3:左调节  0x4:右调节 0x5:停止"
SmartUnloading				:BYTE;	//智能卸料				5	32	2	"0x0:无效  0x1:停止  0x2:开始"

//HU_ControlInformation2	大屏ID2	0x18FF02FE	65280	6	Periodic	100ms	8  FROM 显示屏据

HU_BSDSwitch				:BOOL;		// BSD开关			1	0	1	"0-Inactive 1-Active"
HU_LDWSwitch				:BOOL;		//LDW开关			1	1	1	"0-Inactive 1-Active"
HU_RCWSwitch 				:BOOL;		//	RCW开关			1	2	1	"0-Inactive 1-Active"
HU_AVMSwitchStatus 			:BYTE;		//	AVM按键状态		1	3	2	"0x0:Inactive/Initial value 0x1:Press down 0x2:Lift up"
HU_XAxisPixel 				:DWORD;		//	X轴分辨率/触摸屏width		2	8	12	
HU_YAxisPixel				:DWORD;		//	Y轴分辨率/触摸屏hight		3	20	12	
HU_XAxisPosition			:DWORD;		//	触屏X轴/x坐标				5	32	12	
HU_YAxisPosition			:DWORD;		//	触屏Y轴/y坐标				6	44	12	
HU_PanelStatus				:BYTE;		//	触摸屏状态					8	56	2	"0x0:Inactive/Initial value 0x1:Press down 0x2:Moving 0x3:Lift up"
ControlModeSelection		:BYTE;		//	智能控制方式选择			8	58	2	"0x0:无效 0x1:车载屏控制  0x2:面板控制 0x3:APP控制"
//Reserved	预留		8	60	4	

// HU_ControlInformation2	大屏ID3	0x18FF03FE	65280	6	Periodic	100ms 	8  FROM 显示屏据
TankSpeedInPavingMode		:BYTE;		//		罐速控制铺路模式		1	0	5	"0x0:无效  0x1:1R/min 0x2:2R/min 0x3:3R/min 0x4:4R/min    0xA:10R/min 0xB:11R/min 0x14:20R/min"
GoHome						:BYTE;		//	搅拌车一键复位				1	5	3	"0x0: 无效 0x1:开始  0x2:停止" 
stopSwitch					:BOOL;		//	搅拌车功能急停开关信号		2	8	1	"0x0:无效  0x1:激活"



END_VAR

// MIC7001/Application/10_gvls/GVL_par
{attribute 'qualified_only'}
VAR_GLOBAL
	
	CanWrite102_par_real : ARRAY[0..7] OF REAL;
    	
	
	CanWrite104_par_real : ARRAY[0..7] OF REAL;
 
	CanWrite105_par_real : ARRAY[0..7] OF REAL;
   
	CanWrite106_par_real : ARRAY[0..7] OF REAL;
	
	
	PAR_SET_real : ARRAY[0..20] OF REAL;
	Brake_SET_real : ARRAY[0..22] OF REAL;
	
	PAR_SET_dint : ARRAY[0..20] OF DINT;  //设定参数
	Brake_SET_dint : ARRAY[0..20] OF DINT;  //制动参数
	 
	Vehicle_number:DINT;
	
END_VAR

// MIC7001/Application/06_jt808/programs/prg_gps
PROGRAM prg_gps
VAR  
	filename:STRING(256) := '/tmp/connect_server.txt';
	hFile: RTS_IEC_HANDLE := 0;
	udiOpenError: RTS_IEC_RESULT;
	connect_open_flag :BOOL := TRUE;
	
	gps :Com_gps;
	com_handle :CAA.HANDLE; 
	packGPRMC : nmeaGPRMC;
	buf:STRING(255);
	gps_ok:BOOL := FALSE;
END_VAR

// 判断后端PPP网络是否连通，如果已经连通，则会同步网络时间
IF connect_open_flag THEN
	hFile := sysfileopen(szFile := filename, am := sysfile.AM_READ, pResult:= ADR(udiOpenError));
	IF hFile = RTS_INVALID_HANDLE THEN
		RETURN;
	END_IF
	
	hFile := MIC7001_BASE.close_file(hFile := hFile);
	connect_open_flag := FALSE;
END_IF

gps(xEnable := TRUE, com_hand := com_handle, gps_str => buf); 

nmea_parse_GPRMC(buf, SIZEOF(buf), ADR(packGPRMC));

IF packGPRMC.status = 'A' THEN
	gps_ok := TRUE;
ELSE
	gps_ok := FALSE;
END_IF

END_PROGRAM

// MIC7001/Application/06_jt808/functions/nmea_parse_GPRMC
FUNCTION nmea_parse_GPRMC : bool
VAR_INPUT
    buff : STRING(255);
	buff_sz : DINT;
	pack : POINTER TO nmeaGPRMC;
END_VAR
VAR
	str:STRING(255);
	rc :BOOL;
	checksum : DINT;	
END_VAR

nmea_parse_GPRMC := FALSE;

str := get_sub_string_1(buff, '$$', ',', 1);   //check 'GPRMC'
IF str <> 'GPRMC' THEN
	RETURN;
END_IF

//find time
str := get_sub_string_1(buff, ',', ',', 1);  
IF len(str) < len('hhmmss')  THEN
	RETURN;  //format error	
END_IF
IF NOT nmea_parse_time(str, ADR(pack^.utc)) THEN
	RETURN;
END_IF

//find status
str := get_sub_string_1(buff, ',', ',', 2);  
IF len(str)<1 THEN
	RETURN; //format error
END_IF
pack^.status := str;

//find lat
str := get_sub_string_1(buff, ',', ',', 3);  
IF len(str)<1 THEN
	RETURN; //format error
END_IF
pack^.lat := get_latlon_from_str(str);

//find ns
str := get_sub_string_1(buff, ',', ',', 4); 
IF len(str)<1 THEN
	RETURN; //format error
END_IF
pack^.ns := str;

//find lon
str := get_sub_string_1(buff, ',', ',', 5); 
IF len(str)<1 THEN
	RETURN; //format error
END_IF
pack^.lon := get_latlon_from_str(str);

//find ew
str := get_sub_string_1(buff, ',', ',', 6); 
IF len(str)<1 THEN
	RETURN; //format error
END_IF
pack^.ew := str;

//find speed
str := get_sub_string_1(buff, ',', ',', 7); 
IF len(str)<1 THEN
	RETURN; //format error
END_IF
pack^.speed := STRING_TO_REAL(str)*1.852;  // 节 -> km/h

//find direction
str := get_sub_string_1(buff, ',', ',', 8); 
IF len(str)<1 THEN
	RETURN; //format error
END_IF
pack^.direction := STRING_TO_REAL(str);

//find date
str := get_sub_string_1(buff, ',', ',', 9); 
IF len(str)<1 THEN
	RETURN; //format error
END_IF
IF NOT nmea_parse_date(str, ADR(pack^.utc)) THEN
	RETURN;
END_IF

//find declination
str := get_sub_string_1(buff, ',', ',', 10); 
IF len(str)<1 THEN
	pack^.declination := 0.0;
ELSE
	pack^.declination := STRING_TO_REAL(str);
END_IF

//find declin_ew
str := get_sub_string_1(buff, ',', ',', 11); 
IF len(str)<1 THEN
	RETURN; //format error
END_IF
pack^.declin_ew := str;

//find mode
str := get_sub_string_1(buff, ',', '*', 12); 
IF len(str) < 1 THEN
//	RETURN; // no mode is allowed
ELSE
	pack^.mode := str;
END_IF

//find checksum
str := get_sub_string_1(buff, '*', '$r', 1); 
IF len(str)<1 THEN
	RETURN; //format error
END_IF
checksum := STRING_TO_DINT(str);

nmea_parse_GPRMC := TRUE;

END_FUNCTION

// MIC7001/Application/06_jt808/functions/get_sub_string_1
FUNCTION get_sub_string_1 : STRING(255)
VAR_INPUT
	in_str : STRING(255);
	char_l : STRING(1);
	char_r : STRING(1);
	index : DINT := 1;
END_VAR
VAR
	start : DINT;
	end : DINT;
	sub_str : STRING(255);
	length : DINT;
	i :DINT;
END_VAR

get_sub_string_1 := '';
sub_str := in_str;
i := index;

length := len(sub_str);
start := 0;
end := length+1;

WHILE i > 0 DO
	start := find(sub_str, char_l);
	IF start = 0 THEN
		RETURN;
	END_IF
	sub_str := right(sub_str, DINT_TO_INT(length-start));
	length := len(sub_str);
	i := i - 1;
END_WHILE

end := find(sub_str, char_r);
IF end = 0 THEN
	end := length + 1;
END_IF
get_sub_string_1 := left(sub_str, DINT_TO_INT(end-1));

END_FUNCTION

// MIC7001/Application/06_jt808/functions/nmea_parse_time
FUNCTION nmea_parse_time : BOOL
VAR_INPUT
	str_time:STRING(255);
	p_utc:POINTER TO nmeaTIME;
END_VAR
VAR
	len_str:DINT;
END_VAR

nmea_parse_time := FALSE;

len_str := len(str_time);
IF len_str < len('hhmmss') THEN
	RETURN;  //format error
END_IF

p_utc^.hour := ANY_TO_DINT(left(str_time,2));
p_utc^.minute := ANY_TO_DINT(mid(str_time,2,3));
p_utc^.second := ANY_TO_DINT(mid(str_time,2,5));
IF len_str = len('hhmmss.u') THEN
	p_utc^.hsecond := ANY_TO_DINT(mid(str_time,1,8));
ELSIF len_str = len('hhmmss.uu') THEN
	p_utc^.hsecond := ANY_TO_DINT(mid(str_time,2,8));
ELSIF len_str = len('hhmmss.uuu') THEN
	p_utc^.hsecond := ANY_TO_DINT(mid(str_time,3,8));
ELSE
	//  no hsecond
END_IF

nmea_parse_time := TRUE;

END_FUNCTION

// MIC7001/Application/06_jt808/functions/get_latlon_from_str
FUNCTION get_latlon_from_str : REAL
VAR_INPUT
	str:STRING;
END_VAR

VAR
	temp:REAL;
	d:INT;
	m:REAL;
END_VAR

// lat format:   ddmm.mmmmmm  度度分分.分分分分分分
// lon format:  dddmm.mmmmmm  度度度分分.分分分分分分
   
temp := STRING_TO_REAL(str);
d := ANY_TO_INT(temp/100);
m := temp/100 - d;
m := m/0.6;

get_latlon_from_str := INT_TO_REAL(d)+m;

// 转换为：   度度度.度度度度度度

END_FUNCTION

// MIC7001/Application/06_jt808/functions/nmea_parse_date
FUNCTION nmea_parse_date : BOOL
VAR_INPUT
	str_time:STRING(255);
	p_utc:POINTER TO nmeaTIME;
END_VAR
VAR
	len_str:DINT;
END_VAR

nmea_parse_date := FALSE;

len_str := len(str_time);
IF len_str < len('ddmmyy') THEN
	RETURN;  //format error
END_IF

p_utc^.day := ANY_TO_DINT(left(str_time,2));
p_utc^.month := ANY_TO_DINT(mid(str_time,2,3));
p_utc^.year := ANY_TO_DINT(mid(str_time,2,5));

nmea_parse_date := TRUE;

END_FUNCTION

// MIC7001/Application/06_jt808/functionblocks/Com_gps
FUNCTION_BLOCK Com_gps
VAR_INPUT
	xEnable : BOOL := FALSE;
END_VAR
VAR_IN_OUT
	com_hand: CAA.HANDLE;
END_VAR
VAR_OUTPUT
	xDone : BOOL := FALSE;
	xError :BOOL := FALSE;
	xBusy : BOOL := FALSE;
	gps_str:STRING(255);
END_VAR
VAR
	ton_fb :TON;
	Com1Params: 			ARRAY [1..7] OF COM.PARAMETER;	(* Settings to communicate with 
the COM Port *)
	ComOpen: 				COM.Open;
	ComClose: 				COM.Close;
	ComWrite: 				COM.Write;
	ComRead: 				COM.Read;	
	Rcv_Cnt: 				CAA.SIZE;
	xCom1CloseError: 		BOOL;
	xCom1WriteError: 		BOOL;
	xCom1ReadError: 		BOOL;
	uiComState: INT := 0;
	ComID:USINT:=5;   //ttymxc4
	position :INT := 0;
	at_cmd :STRING := 'AT$r';
	at_buffer :STRING;
	ate0_cmd :STRING := 'ATE0$r';
	ate0_buffer :STRING;
	csq_cmd :STRING := 'AT+CSQ$r';
	csq_buffer :STRING;
	
	accid_cmd :STRING := 'AT+ICCID$r';
	iccid_read_buffer :STRING(255);
	ICCID_HEAD:STRING := '+ICCID: ';
	iccid:STRING(32);
	
	lac:STRING(4) := '0000';
	ci :STRING(4) := '0000';
	lac_set_cmd :STRING := 'AT+CREG=2$r';
	lac_read_cmd :STRING(255);
	
	
	lac_get_cmd :STRING := 'AT+CREG?$r';
	lac_read_buffer :STRING(255);
	
	lac_close_cmd :STRING := 'AT+CREG=0$r';
	lac_close_buffer :STRING(255);
	
	LACID_HEAD:STRING := '+CREG:';
	lac_str:STRING(8);
	ci_str:STRING(8);
	
	at_GPSCLOSE_buffer :STRING(255);
	at_GPSCLOSE_cmd :STRING := 'AT+QGPS=0$r';    
	at_GPSOPEN_cmd :STRING := 'AT+QGPS=1$r';     
	at_GPSOPEN_buffer :STRING(255);
	
	at_GPSSET_cmd :STRING := 'AT+QGPSCFG="nmeasrc",1$r';     
	at_GPSSET_buffer :STRING(255);
	
	at_GPSREAD_cmd :STRING := 'AT+QGPSGNMEA="RMC"$r';    
	at_GPSREAD_buffer :STRING(255);
	
	at_ask_buffer3 :STRING(1000);
	bit_start:INT;
	bit_end:INT;
	bit_start1:INT;
	bit_end1:INT;
	jd_info:STRING;
	wd_info:STRING;
	jd:REAL;
	wd:REAL;
	R_TIME:TIME;
	
	xDone_internal : BOOL := FALSE;
	xError_internal :BOOL := FALSE;
	
	sudu_info :STRING;
	bit_end2:INT;
	sd:REAL;
	
	ton_err:ton;
	cntr_40:DINT := 0;
END_VAR

IF NOT xEnable THEN
	xDone := FALSE;
	xError := FALSE;
	xBusy := FALSE;
	uiComState := 0;
	RETURN;
END_IF

CASE uiComState OF
	0:
	Com1Params[1].udiParameterId := COM.CAA_Parameter_Constants.udiPort;
	Com1Params[1].udiValue := ComID; 
	Com1Params[2].udiParameterId := COM.CAA_Parameter_Constants.udiBaudrate;
	Com1Params[2].udiValue := 115200;
	Com1Params[3].udiParameterId := COM.CAA_Parameter_Constants.udiParity;
	Com1Params[3].udiValue := INT_TO_UINT(COM.PARITY.NONE);
	Com1Params[4].udiParameterId := COM.CAA_Parameter_Constants.udiStopBits;
	Com1Params[4].udiValue := INT_TO_UINT(COM.STOPBIT.ONESTOPBIT);
	Com1Params[5].udiParameterId := COM.CAA_Parameter_Constants.udiTimeout;
	Com1Params[5].udiValue := 0;
	Com1Params[6].udiParameterId := COM.CAA_Parameter_Constants.udiByteSize;
	Com1Params[6].udiValue := 8;
	Com1Params[7].udiParameterId := COM.CAA_Parameter_Constants.udiBinary;
	Com1Params[7].udiValue := 0;					
	ComOpen(xExecute := TRUE, usiListLength:=UINT_TO_USINT(SIZEOF(Com1Params)/SIZEOF(COM.PARAMETER)),pParameterList:= ADR(Com1Params),hCom=> com_hand);			
	IF ComOpen.xError THEN
		ton_err(in := FALSE, pt := T#5S);
		uiComState := 32767;
	ELSIF ComOpen.xDone THEN
		uiComState := 1;
		com_hand := ComOpen.hCom;
		ComWrite(xExecute := FALSE,hCom:= com_hand);	
		ComRead(xExecute := FALSE,hCom:= com_hand);
	END_IF
	
	1:  // write "AT\r"
	ComWrite(xExecute := TRUE,hCom:= com_hand,pBuffer:= ADR(at_cmd),szSize:=len(at_cmd));		
	IF ComWrite.xError THEN
		uiComState := 200;
	END_IF
	IF ComWrite.xDone THEN
		ComWrite(xExecute := FALSE, hCom:= com_hand);
		uiComState := 2;
	END_IF
	
	2:
	ton_fb(IN := TRUE, PT := TIME#300MS);
	IF (ton_fb.Q) THEN
		ton_fb(IN := FALSE, PT := TIME#300MS);
		uiComState := 3;
	END_IF
	
	3:
	ComRead(xExecute := TRUE,hCom:= com_hand, pBuffer:= ADR(at_buffer), szBuffer:= SIZEOF(at_buffer));			
	IF ComRead.xError THEN
		uiComState := 32767;
	END_IF
	IF ComRead.xDone THEN
		position := find(at_buffer, 'OK');
		IF position > 0 THEN
			uiComState := 10;
		ELSE
			uiComState := 200;
		END_IF
		ComRead(xExecute := FALSE, hCom:= com_hand);
	END_IF
	
(*	
	4: // write "ATE0\r"
	ComWrite(xExecute := TRUE,hCom:= com_hand,pBuffer:= ADR(ate0_cmd),szSize:=len(ate0_cmd));		
	IF ComWrite.xError THEN
		uiComState := 200;
	END_IF
	IF ComWrite.xDone THEN
		ComWrite(xExecute := FALSE, hCom:= com_hand);
		uiComState := 5;
	END_IF
	
	5:
	ton_fb(IN := TRUE, PT := TIME#300MS);
	IF (ton_fb.Q) THEN
		ton_fb(IN := FALSE, PT := TIME#300MS);
		uiComState := 6;
	END_IF
	
	6:
	ComRead(xExecute := TRUE,hCom:= com_hand, pBuffer:= ADR(ate0_buffer), szBuffer:= SIZEOF(ate0_buffer));			
	IF ComRead.xError THEN
		uiComState := 200;
	END_IF
	IF ComRead.xDone THEN
		position := find(ate0_buffer, 'OK');
		IF position > 0 THEN
			uiComState := 10;
		ELSE
			uiComState := 200;
		END_IF
		ComRead(xExecute := FALSE, hCom:= com_hand);
	END_IF
	*)
	
	
	10: // write "AT+CSQ\r"
	ComWrite(xExecute := TRUE,hCom:= com_hand,pBuffer:= ADR(csq_cmd),szSize:=len(csq_cmd));		
	IF ComWrite.xError THEN
		uiComState := 200;
	END_IF
	IF ComWrite.xDone THEN
		ComWrite(xExecute := FALSE, hCom:= com_hand);
		uiComState := 11;
	END_IF
	
	11:
	ton_fb(IN := TRUE, PT := TIME#300MS);
	IF (ton_fb.Q) THEN
		ton_fb(IN := FALSE, PT := TIME#300MS);
		uiComState := 12;
	END_IF
	
	12:
	ComRead(xExecute := TRUE,hCom:= com_hand, pBuffer:= ADR(csq_buffer), szBuffer:= SIZEOF(csq_buffer));			
	IF ComRead.xError THEN
		uiComState := 200;
	END_IF
	IF ComRead.xDone THEN
		position := find(csq_buffer, 'OK');
		IF position > 0 THEN
			uiComState := 13;
		ELSE
			uiComState := 200;
		END_IF
		ComRead(xExecute := FALSE, hCom:= com_hand);
	END_IF
	
	13:
	ComWrite(xExecute := TRUE,hCom:= com_hand,pBuffer:= ADR(accid_cmd),szSize:=len(accid_cmd));		
	IF ComWrite.xError THEN
		uiComState := 200;
	END_IF
	IF ComWrite.xDone THEN
		ComWrite(xExecute := FALSE, hCom:= com_hand);
		uiComState := 14;
	END_IF
	
	14:
	ton_fb(IN := TRUE, PT := TIME#300MS);
	IF (ton_fb.Q) THEN
		ton_fb(IN := FALSE, PT := TIME#300MS);
		uiComState := 15;
	END_IF
	
	15:
	ComRead(xExecute := TRUE,hCom:= com_hand, pBuffer:= ADR(iccid_read_buffer), szBuffer:= SIZEOF(iccid_read_buffer));			
	IF ComRead.xError THEN
		uiComState := 200;
	END_IF
	IF ComRead.xDone THEN
		IF ComRead.szsize > 0 THEN
			position := find(iccid_read_buffer, ICCID_HEAD);
			IF position > 0 THEN
				iccid := mid(iccid_read_buffer, 20, position + len(ICCID_HEAD));
				uiComState := 16;
			ELSE
				uiComState := 200;
			END_IF
		ELSE
			uiComState := 200;
		END_IF
		ComRead(xExecute := FALSE, hCom:= com_hand);
	END_IF
	
	16:
	ComWrite(xExecute := TRUE,hCom:= com_hand,pBuffer:= ADR(at_GPSCLOSE_cmd),szSize:=len(at_GPSCLOSE_cmd));		
	IF ComWrite.xError THEN
		uiComState := 200;
	END_IF
	IF ComWrite.xDone THEN
		ComWrite(xExecute := FALSE, hCom:= com_hand);
		uiComState := 17;
	END_IF
	
	17:
	ton_fb(IN := TRUE, PT := TIME#300MS);
	IF (ton_fb.Q) THEN
		ton_fb(IN := FALSE, PT := TIME#300MS);
		uiComState := 18;
	END_IF
	
	18:
	ComRead(xExecute := TRUE,hCom:= com_hand, pBuffer:= ADR(at_GPSCLOSE_buffer), szBuffer:= SIZEOF(at_GPSCLOSE_buffer));			
	IF ComRead.xError THEN
		uiComState := 200;
	END_IF
	IF ComRead.xDone THEN
		uiComState := 25;
		ComRead(xExecute := FALSE, hCom:= com_hand);
	END_IF
	
	25:
	ComWrite(xExecute := TRUE,hCom:= com_hand,pBuffer:= ADR(at_GPSOPEN_cmd),szSize:= len(at_GPSOPEN_cmd));		
	IF ComWrite.xError THEN
		uiComState := 200;
	END_IF
	IF ComWrite.xDone THEN		
		ComWrite(xExecute := FALSE);
		uiComState := 26;
	END_IF
	
	26:
	ton_fb(IN := TRUE, PT := TIME#300MS);
	IF (ton_fb.Q) THEN
		ton_fb(IN := FALSE, PT := TIME#300MS);
		uiComState := 27;
	END_IF

	27:
	ComRead(xExecute := TRUE,hCom:= com_hand, pBuffer:= ADR(at_GPSOPEN_buffer), szBuffer:= SIZEOF(at_GPSOPEN_buffer));			
	IF ComRead.xError THEN
		uiComState := 200;
	END_IF
	IF ComRead.xDone THEN
		position := find(at_GPSOPEN_buffer, 'OK');
		IF position > 0 THEN
			uiComState := 28;
		ELSE
			uiComState := 200;
		END_IF
		ComRead(xExecute := FALSE, hCom:= com_hand);
	END_IF
	
	
	28:
	ComWrite(xExecute := TRUE,hCom:= com_hand,pBuffer:= ADR(at_GPSSET_cmd),szSize:= len(at_GPSSET_cmd));		//发送AT指令，查询获取的经纬度
	IF ComWrite.xError THEN
		uiComState := 200;
	END_IF
	IF ComWrite.xDone THEN		
		ComWrite(xExecute := FALSE);
		uiComState := 29;
	END_IF
	
	29:
	ton_fb(IN := TRUE, PT := TIME#300MS);
	IF (ton_fb.Q) THEN
		ton_fb(IN := FALSE, PT := TIME#300MS);
		uiComState := 30;
	END_IF
	
	30:
	ComRead(xExecute := TRUE,hCom:= com_hand, pBuffer:= ADR(at_GPSSET_buffer), szBuffer:= SIZEOF(at_GPSSET_buffer));			
	IF ComRead.xError THEN
		uiComState := 200;
	END_IF
	IF ComRead.xDone THEN
		position := find(at_GPSSET_buffer, 'OK');
		IF position > 0 THEN
			uiComState := 31;
		ELSE
			uiComState := 200;
		END_IF
		ComRead(xExecute := FALSE, hCom:= com_hand);
	END_IF
	
	
	31:
	ComWrite(xExecute := TRUE,hCom:= com_hand,pBuffer:= ADR(at_GPSREAD_cmd),szSize:= len(at_GPSREAD_cmd));		//发送AT指令，查询获取的经纬度
	IF ComWrite.xError THEN
		uiComState := 200;
	END_IF
	IF ComWrite.xDone THEN		
		ComWrite(xExecute := FALSE);
		uiComState := 32;
	END_IF

	32:
	ton_fb(IN := TRUE, PT := TIME#300MS);
	IF (ton_fb.Q) THEN
		ton_fb(IN := FALSE, PT := TIME#300MS);
		uiComState := 33;
	END_IF
	
	33:
	ComRead(xExecute := TRUE,hCom:= com_hand, pBuffer:= ADR(at_GPSREAD_buffer), szBuffer:= SIZEOF(at_GPSREAD_buffer));
	IF ComRead.xError THEN
		uiComState := 200;
	END_IF
    IF ComRead.xDone THEN
		gps_str := at_GPSREAD_buffer;
		uiComState := 40;
		cntr_40 := 0;
		ComRead(xExecute := FALSE, hCom:= com_hand);
	END_IF
	
	40:  // waiting
	   cntr_40 := cntr_40+1;
	   IF cntr_40 > 20 THEN // 2s
		   uiComState := 31;
	   END_IF
	
	200:
		xError_internal := TRUE;
		uiComState := 202;
		
	201:
		xDone_internal := TRUE;
		uiComState := 202;
		
	202:
		ComClose(xExecute := FALSE, hCom:= com_hand); 	
		uiComState := 203;
	
	203:
		ComClose(xExecute := TRUE,hCom:= com_hand);
		IF ComClose.xError THEN
			uiComState := 32767;
		END_IF
		
		IF ComClose.xDone THEN
			ComClose(xExecute := FALSE, hCom:= com_hand); 	
		
			IF xDone_internal THEN
				uiComState := 255;
			END_IF
			
			IF xError_internal THEN
				uiComState := 32767;
			END_IF
		END_IF
	
	
	255:
		xDone := TRUE;
		
	32767:	
		xError := TRUE;
		ton_err(in := TRUE, pt := T#5S);
		IF ton_err.Q THEN
			ComOpen(xExecute := FALSE, usiListLength:=UINT_TO_USINT(SIZEOF(Com1Params)/SIZEOF(COM.PARAMETER)),pParameterList:= ADR(Com1Params),hCom=> com_hand);	
			ton_err(in := FALSE, pt := T#5S);
			uiComState := 0;
		END_IF
END_CASE

END_FUNCTION_BLOCK

// MIC7001/Application/06_jt808/programs/prg_jt808
PROGRAM prg_jt808
VAR
	inited : BOOL := FALSE;
	fluidLow:INT := 0;
	lossWater:INT := 0;
	dirtyWater:INT := 0;
	littleWater:INT := 0;
	pressSuper:INT := 0;
	
	strShmFileDown : STRING := 'SHM_JT808_DW_7001';
	strShmFileUp : STRING := 'SHM_JT808_UP_7001';
	hShMemDown: RTS_IEC_HANDLE := RTS_INVALID_HANDLE ;
	hShMemUp: RTS_IEC_HANDLE := RTS_INVALID_HANDLE ;
	ResultRead: RTS_IEC_RESULT;
	ResultWrite: RTS_IEC_RESULT;
	
	iRead: __UXINT;
	iWrite: __UXINT;
	shmDataDown:stShmJT808Down;
	shmDataUp:stShmJT808Up;
	sizeOfStFromAliyun:__UXINT := SIZEOF(stShmJT808Down);
	sizeOfStToAliyun:__UXINT := SIZEOF(stShmJT808Up);
	
	sim_data : DINT := 0;
	digi_val :DWORD := 0;
	lock_1 :BOOL := FALSE;
	lock_2 :BOOL := FALSE;
	unlock :BOOL := FALSE;
	test_val2 :DINT;
	
	get_dt:dtu.GetDateandTime();
	tempdt : DWORD;
	g_uiYear:UINT;
	g_uiMonth:UINT;
	g_uiDate:UINT;
	g_uiHour:UINT;
	g_uiMinute:UINT;
	g_uiSecond:UINT;
END_VAR


IF NOT inited THEN
 	IF NOT init() THEN  // 初始化失败
		RETURN;
	ELSE
		inited := TRUE;
		
		sim_data := 0;
		test_val2 := 0;
	END_IF  
END_IF

IF read_from_server() THEN
   // 读取阿里云发来的数据
	IF shmDataDown.ctrl > 0 THEN
		// 处理命令通道1
	END_IF
END_IF

// 准备上传到阿里云的数据
sim_data := sim_data + 1;

get_dt(xExecute := TRUE);
 IF get_dt.xDone THEN
  tempdt := DT_TO_DWORD(get_dt.dtDateandtime);
  tempdt := tempdt + 3600*8;   // utc 时间转为北京时间
  dtu.DTSplit(DWORD_TO_DT(tempdt), ADR(g_uiYear), ADR(g_uiMonth), ADR(g_uiDate), ADR(g_uiHour), ADR(g_uiMinute), ADR(g_uiSecond));

  get_dt(xExecute := FALSE);

 END_IF

shmDataUp.location.asc_time[0] := ANY_TO_BYTE(g_uiYear MOD 100);
shmDataUp.location.asc_time[1] := ANY_TO_BYTE(g_uiMonth);
shmDataUp.location.asc_time[2] := ANY_TO_BYTE(g_uiDate);
shmDataUp.location.asc_time[3] := ANY_TO_BYTE(g_uiHour);
shmDataUp.location.asc_time[4] := ANY_TO_BYTE(g_uiMinute);
shmDataUp.location.asc_time[5] := ANY_TO_BYTE(g_uiSecond);

shmDataUp.loc_ext.km_all := ANY_TO_DINT( gvl_es.trip_all_1939*10);      // jt808 unit: 0.1Km
shmDataUp.loc_ext.fuel_trip := ANY_TO_DINT(gvl_es.fuel_trip_engine*2);  // jt808 unit: 0.5L
shmDataUp.loc_ext.fuel_all := ANY_TO_DINT( gvl_es.fuelall_engine*2);    // jt808 unit: 0.5L
shmDataUp.loc_ext.fuel_r_h := ANY_TO_DINT(gvl_es.fuelrate_engine*20);   // jt808 unit: 0.05L/h
IF gvl_es.fuel_100km = 0 OR gvl_es.fuel_100km = 999 THEN
	shmDataUp.loc_ext.fuel_r_l := 0;
ELSE
	shmDataUp.loc_ext.fuel_r_l := ANY_TO_DINT(512*100/gvl_es.fuel_100km);   // jt808 unit: 1/512Km/L
END_IF

IF prg_gps.packGPRMC.status = 'A' THEN  // GPS定位成功
	shmDataUp.location.latitude := ANY_TO_DINT(prg_gps.packGPRMC.lat*1000000);
	shmDataUp.location.longitude := ANY_TO_DINT(prg_gps.packGPRMC.lon*1000000);
	shmDataUp.location.altitude := 54;
	shmDataUp.location.speed := ANY_TO_INT(prg_gps.packGPRMC.speed);
	shmDataUp.location.bearing := ANY_TO_INT(prg_gps.packGPRMC.direction);
	shmDataUp.location.status := 16#03;   
ELSIF 	prg_gps.packGPRMC.status = 'V' THEN  // 有GPS，但尚未定位成功
	shmDataUp.location.latitude := 0;
	shmDataUp.location.longitude := 0;	
	shmDataUp.location.altitude := 0;
	shmDataUp.location.speed := 0;
	shmDataUp.location.bearing := 0;	
	shmDataUp.location.status := 16#02;   
ELSE	// 没有GPS
    shmDataUp.loc_ext.lac := MIC7001_base.read_num_from_file(filename := '/tmp/lac.txt');
	shmDataUp.loc_ext.cid := MIC7001_base.read_num_from_file(filename := '/tmp/cid.txt');
	shmDataUp.location.latitude := 28230306;
	shmDataUp.location.longitude := 113414176;	
	shmDataUp.location.altitude := 0;	
	shmDataUp.location.status := 16#03;   
END_IF

IF send_to_server() THEN
	// write ok
END_IF

METHOD send_to_server : bool
VAR_INPUT
END_VAR
send_to_server := FALSE;

iWrite := sysshm.SysSharedMemoryWrite(hShMemUp, 0, ADR(shmDataUp), sizeOfStToAliyun, ADR(ResultWrite));
IF iWrite = sizeOfStToAliyun THEN
	send_to_server := TRUE;
END_IF

RETURN;
END_METHOD

METHOD read_from_server : bool
VAR_INPUT
END_VAR
read_from_server := FALSE;

iRead := sysshm.SysSharedMemoryRead(hShMemDown, 0, ADR(shmDataDown), sizeOfStFromAliyun, ADR(ResultRead));
IF iRead = sizeOfStFromAliyun THEN
    read_from_server := TRUE;
END_IF

RETURN;
END_METHOD

METHOD init : bool
VAR_INPUT
END_VAR
init := FALSE;

IF hShMemDown = RTS_INVALID_HANDLE  THEN
	hShMemDown := sysshm.SysSharedMemoryCreate(strShmFileDown, 0, ADR(sizeOfStFromAliyun), ADR(ResultRead));	
END_IF

IF hShMemUp = RTS_INVALID_HANDLE  THEN
	hShMemUp := sysshm.SysSharedMemoryCreate(strShmFileUp, 0, ADR(sizeOfStToAliyun), ADR(ResultRead));	
END_IF

IF hShMemDown = RTS_INVALID_HANDLE  OR hShMemUp = RTS_INVALID_HANDLE  THEN
	RETURN;
END_IF

init := TRUE;
RETURN;
END_METHOD

END_PROGRAM
